Yaskawa INFORM job: MTFTEST2.JBI

/JOB
//NAME MTFTEST2
//POS
///NPOS 1,1,0,1,0,0
///TOOL 0
///POSTYPE ROBOT
///RECTAN
///RCONF 0,0,0,0,0,0,0,0,0,0,0,0,0,0,0,0,0,0,0,0,0,0,0,0
C00000=412.405,-1517.658,-1319.175,-20.9817,4.8842,-3.0056
BC00000=247.717,3642.643,1999.610
///POSTYPE BASE
P00007=759.319,2124.985,680.441,-20.9817,4.8842,-3.0056
//INST
///DATE 2024/01/24 13:09
///ATTR SC,RW,RJ
////FRAME ROBOT
///GROUP1 RB1,BS1
NOP
REFP 6 C00000 BC00000
CALL JOB:MTFTEST ARGF7
PAUSE
MOVJ P007 VJ=50.00
END
